% RSLogix 500 project I2P JOB 21 - ANDREW_HOEMMEN_BAK065.RSS, saved by version 10.00.00.00 %
PROJECT "ML03A"    % processor: Bul.1763 MicroLogix 1100 Series B %

PROGRAM FILES
  LAD 2   5 rungs

DATA FILES
  O0 OUTPUT  4 elements
  I1 INPUT  6 elements
  S2 STATUS  66 elements
  B3 BINARY  1 elements
  T4 TIMER  1 elements
  C5 COUNTER  1 elements
  R6 CONTROL  1 elements
  N7 INTEGER  1 elements
  F8 FLOAT  1 elements

LADDER 2
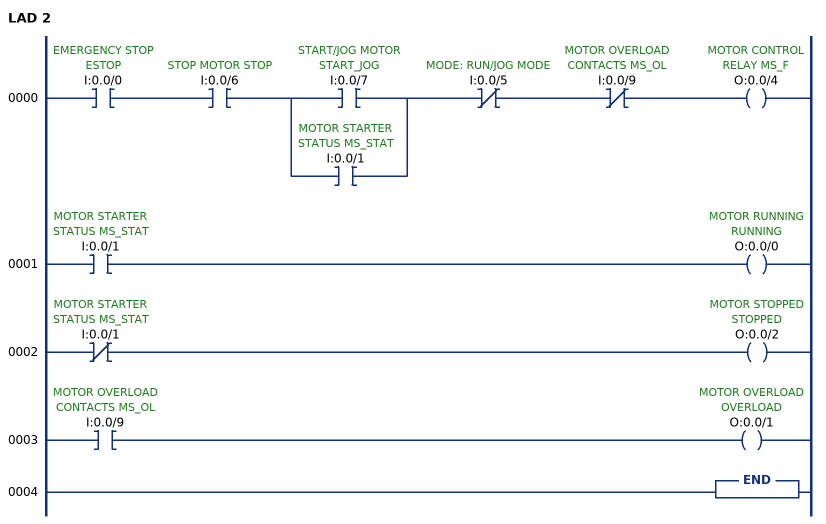
% Rung: 0 %
SOR XIC I:0.0/0 XIC I:0.0/6 BST XIC I:0.0/7 NXB XIC I:0.0/1 BND XIO I:0.0/5 XIO I:0.0/9 OTE O:0.0/4 EOR
%   I:0.0/0  ESTOP  "EMERGENCY STOP" %
%   I:0.0/6  STOP  "STOP MOTOR" %
%   I:0.0/7  START_JOG  "START/JOG MOTOR" %
%   I:0.0/1  MS_STAT  "MOTOR STARTER STATUS" %
%   I:0.0/5  MODE  "MODE: RUN/JOG" %
%   I:0.0/9  MS_OL  "MOTOR OVERLOAD CONTACTS" %
%   O:0.0/4  MS_F  "MOTOR CONTROL RELAY" %
% Rung: 1 %
SOR XIC I:0.0/1 OTE O:0.0/0 EOR
%   I:0.0/1  MS_STAT  "MOTOR STARTER STATUS" %
%   O:0.0/0  RUNNING  "MOTOR RUNNING" %
% Rung: 2 %
SOR XIO I:0.0/1 OTE O:0.0/2 EOR
%   I:0.0/1  MS_STAT  "MOTOR STARTER STATUS" %
%   O:0.0/2  STOPPED  "MOTOR STOPPED" %
% Rung: 3 %
SOR XIC I:0.0/9 OTE O:0.0/1 EOR
%   I:0.0/9  MS_OL  "MOTOR OVERLOAD CONTACTS" %
%   O:0.0/1  OVERLOAD  "MOTOR OVERLOAD" %
% Rung: 4 %
SOR END EOR

OTHER DOCUMENTED ADDRESSES
  B3:0/0  STOP_BIT  "STOP BIT"
  B3:0/1  FWD_BIT  "FORWARD BIT"
  B3:0/2  FWD_JOG  "FORWARD JOG BIT"
  B3:0/3  REV_BIT  "REVERSE BIT"
  B3:0/4  REV_JOG  "REVERSE JOG"
  B3:0/5  CHAN_BIT  "CHANGING BIT"
  B3:0/6  LAST_FWD  "LAST FORWARD"
  B3:0/7  LAST_REV  "LAST REVERSE"
  DIR_STATS  
  I:0.0/2  DIR_STAT
  I:0.0/3  MODE_AUTO  "MODE ON/OFF AUTO"
  I:0.0/4  3PSS_B  "3PSS B"
  I:0.0/8  JOG  "JOG MOTOR"
  O:0.0/3  FULL  "TANK FULL"
  O:0.0/5  CR2  "DIRECTION CONTROL RELAY 2"
  T4:0.ACC  BLINK  "LIGHT BLINKING"

DATA TABLE (non-zero values as saved)
DATA T4
% .PRE .ACC %
% T4:0 % 8 0
